// TIA Portal V17 export
// export: Created 2022-07-28T18:03:17.298759Z, ExportSetting None, DisplayName Totally Integrated Automation Portal, DisplayVersion V17, DisplayName TIA Portal Openness, DisplayVersion V17, DisplayName TIA Portal Teamcenter Gateway, DisplayVersion V17, DisplayName TIA Portal Version Control Interface, DisplayVersion V17, DisplayName TIA Portal Test Suite Advanced, DisplayVersion V17, DisplayName SINAMICS Startdrive Advanced, DisplayVersion V17, DisplayName SINAMICS DCC, DisplayVersion V17, DisplayName SINAMICS Startdrive G130, G150, S120, S150, SINAMICS MV, S210, DisplayVersion V17, DisplayName SINAMICS Startdrive G110M, G120, G120C, G120D, G120P, G115D, DisplayVersion V17, DisplayName STEP 7 Professional, DisplayVersion V17, DisplayName SIMATIC Energy Suite, DisplayVersion V17, DisplayName STEP 7 CFC, DisplayVersion V17, DisplayName STEP 7 Safety, DisplayVersion V17, DisplayName WinCC Advanced / Unified PC, DisplayVersion V17, DisplayName SIMATIC Visualization Architect, DisplayVersion V17
TYPE "_Inverter_352Tel_STW_Bits"
   STRUCT
      ReadyToSwitchOn : Bool;   // Bit 0 - 1 = Ready for switched on; electronics initialized; pulses locked
      ReadyToOperation : Bool;   // Bit 1 - 1 = Ready for operation. Start as soon as ON1 is active (bit 0 = 1 in CTW)
      OperationEnabled : Bool;   // Bit 2 - 1 = Motor follows setpoint
      FaultActive : Bool;   // Bit 3 - 1 = Fault present. Acknowlege is requaired
      OFF2Inactive : Bool;   // Bit 4 - 0 = OFF2 is inactive
      OFF3Inactive : Bool;   // Bit 5 - 0 = OFF3 is inactive
      LockoutActive : Bool;   // Bit 6 - 1 = Lockout active. Motor switched on after trig ON1
      AlarmActive : Bool;   // Bit 7 - 1 = Alarm is active. Acknowlege not requaired
      SetpointReached : Bool;   // Bit 8 - 1 = Setpoint speed is achived
      CtrlRequest : Bool;   // Bit 9 - 1 = The automation system is requested to assume control
      MaxSpeedReached : Bool;   // Bit 10 - 1 = Actual speed greater or equal to maximum speed
      IMP_LimitReached : Bool;   // Bit 11 - 0 = Current, torque or power limit has been reached or exceeded
      BrakeOpen : Bool;   // Bit 12 - 1 = Signal to open motor holding brake
      Overtemperature : Bool;   // Bit 13 - 0 = Alarm motor overtemperature
      ForwardBeckward : Bool;   // Bit 14 - 1 = Motor rotates forwards (act>0); 0 = Motor rotates backwards (act<0)
      PowerUnitOverload : Bool;   // Bit 15 - 1 = No alarm, thermal power unit overload
   END_STRUCT;
END_TYPE
